// TIA Portal V19 export
DATA_BLOCK "Send to AlcipM3"   // DB476
TITLE = Send Interface to Flex A AlcipM3
{ S7_Optimized_Access := 'TRUE' }
// stored: AutoNumber false, MemoryReserve 0
   VAR RETAIN
      CC1 : Struct   // Polygon Filler
         CC_CL_RemWdCnt : Int;   // Watchdog Counter
         CC_CL_Eng_bit : Bool;
         CC_CL_LyeReq : Bool;
         CC_CL_AcidReq : Bool;
         CC_CL_WaterReq : Bool;
         CC_CL_RinseW_Req : Bool;
         CC_CL_LyeReturn : Bool;
         CC_CL_AcidReturn : Bool;
         CC_CL_RinseW_Return : Bool;
         CC_CL_ObjNoReturn : Bool;
         CC_CL_HeatingReq : Bool;
         CC_CL_ObjEn : Bool;
         CC_CL_ObjReady : Bool;
         CC_CL_RinseP_Return : Bool;
         CC_CL_Start : Bool;
         CC_CL_ObjWd : Bool;
         CC_CL_CipTerminated : Bool;
         CC_CL_spare1 : Bool;
         CC_CL_spare2 : Bool;
         CC_CL_spare3 : Bool;
         CC_CL_spare4 : Bool;
         CC_CL_spare5 : Bool;
         CC_CL_spare6 : Bool;
         CC_CL_spare7 : Bool;
         CC_CL_spare8 : Bool;
         CC_CL_spare9 : Bool;
         CC_CL_spare10 : Bool;
         CC_CL_spare11 : Bool;
         CC_CL_spare12 : Bool;
         CC_CL_spare13 : Bool;
         CC_CL_spare14 : Bool;
         CC_CL_spare15 : Bool;
         CC_CL_spare16 : Bool;
      END_STRUCT;
      hmi : Struct
         commsFault : Bool;
         s1 : Bool;   // spare
         s2 : Bool;   // spare
         s3 : Bool;   // spare
         s4 : Bool;   // spare
         s5 : Bool;   // spare
         s6 : Bool;   // spare
         s7 : Bool;   // spare
         s8 : Bool;   // spare
         s9 : Bool;   // spare
         s10 : Bool;   // spare
         s11 : Bool;   // spare
         s12 : Bool;   // spare
         s13 : Bool;   // spare
         s14 : Bool;   // spare
         s15 : Bool;   // spare
      END_STRUCT;
      _word2 : Word;
      _word3 : Word;
      _word4 : Word;
      _word5 : Word;
   END_VAR
BEGIN
END_DATA_BLOCK
